PROGRAM MAIN
VAR
	fbTest : Fb_test;
END_VAR

//Test first commit
fbTest();

END_PROGRAM

(* stored: Version 1.1.0.1, ProductVersion 3.1.4024.12
   POU MAIN: Id {a797216d-7fab-49e4-8fc0-a11a48df1647}, SpecialFunc None *)
